{attribute 'qualified_only'}
VAR_GLOBAL
END_VAR

(* stored: Version 1.1.0.1, ProductVersion 3.1.4024.4
   GVL STATE: Id {2a284180-e1f9-480f-95fa-305b8cc46bee} *)
